INTERFACE ITimeoutException EXTENDS IGeneralException

METHOD Throw
VAR_INPUT
	sourceNamespaceName : STRING;
	sourceClassName : STRING;
	sourcePOUName : STRING;
	sourcePosition : STRING;
	timeoutValue : TIME;
	operationName : WSTRING := "";
END_VAR
END_METHOD

END_INTERFACE

(* stored: Version 1.1.0.1
   Itf ITimeoutException: Id {ac6243fb-9a96-4392-a8e2-9c8ccc7744cc}
   Method Throw: Id {f86ea1ff-ed67-4ee6-9653-f2452f2af1f0} *)
